PROGRAM BackgroundRS232
VAR
END_VAR

BackgroundEL6001();

END_PROGRAM

(* stored: Version 1.1.0.1, ProductVersion 3.1.4024.12
   POU BackgroundRS232: Id {a474ab24-92b2-4faa-ab36-f1eb12602ab9}, SpecialFunc None *)
